FUNCTION_BLOCK EL1134
VAR
	_io : EL1xx4_Data;
	{attribute addProperty Name "WcState"}
	_wcState : WcStateInputToggle;
	{attribute addProperty Name "Info data"}
	_infoData : InfoDataBase;
END_VAR

PROPERTY IO : REFERENCE TO EL1xx4_Data
GET
IO REF= _io;
END_GET
END_PROPERTY

PROPERTY WcState : REFERENCE TO WcStateInputToggle
GET
WcState REF= _wcState;
END_GET
END_PROPERTY

END_FUNCTION_BLOCK

(* stored: Version 1.1.0.1, ProductVersion 3.1.4024.9
   POU EL1134: Id {34a828e5-990d-07d9-0523-33815c573a20}, SpecialFunc None
   Property IO: Id {725f12bb-c990-0461-25cf-63a119fb7ed0}
   Get Get: Id {0de7c1b2-c705-0de9-27c8-66b06f88e516}
   Property WcState: Id {3ef4a88d-2586-033a-0ca6-1d224191e882}
   Get Get: Id {98e392d7-9384-0d49-0538-315bddfbce29} *)
